// TIA Portal V16 export
// export: Created 2024-12-03T15:41:45.1410712Z, ExportSetting WithReadOnly, DisplayName Totally Integrated Automation Portal, DisplayVersion V16 Update 6, DisplayName TIA Portal Version Control Interface, DisplayVersion V16 Update 2, DisplayName TIA Portal Openness, DisplayVersion V16 Update 6, DisplayName TIA Portal Teamcenter Gateway, DisplayVersion V16, DisplayName SINAMICS Startdrive Advanced, DisplayVersion V16 Update 5, DisplayName SINAMICS Startdrive G130, G150, S120, S150, SINAMICS MV, S210, DisplayVersion V16 Update 5, DisplayName SINAMICS Startdrive G110M, G120, G120C, G120D, G120P, G115D, DisplayVersion V16 Update 5, DisplayName STEP 7 Professional, DisplayVersion V16 Update 6, DisplayName STEP 7 Safety, DisplayVersion V16, DisplayName WinCC Advanced / Unified PC, DisplayVersion V16 Update 6
TYPE "IT2000M_Scale_IN_UDT"
// stored: CreationDate 2021-07-13T07:41:36.2278727Z, InterfaceModifiedDate 2021-07-11T06:56:03.4750348Z, IsConsistent true, LibraryConformanceStatus The object is library-conformant., ModifiedDate 2021-07-11T06:56:03.4750348Z
   STRUCT
      Inputs : Struct
         spare : Byte;
         spare_0 : Bool;
         spare_1 : Bool;
         spare_2 : Bool;
         spare_3 : Bool;
         spare_4 : Bool;
         spare_5 : Bool;
         Input_E0 : Bool;
         Input_E1 : Bool;
      END_STRUCT;
      Outputs : Struct
         spare : Byte;
         spare_0 : Bool;
         spare_1 : Bool;
         spare_2 : Bool;
         spare_3 : Bool;
         spare_4 : Bool;
         spare_5 : Bool;
         Output_A0 : Bool;
         Output_A1 : Bool;
      END_STRUCT;
      NetWeight : Int;
      GrossWeight : Int;
      Status : Struct
         Handshake : Bool;
         Status : Bool;   // 1 = command carried out
         OutOfTolerance : Bool;
         FlowRateLow : Bool;
         spare_0 : Bool;
         spare_1 : Bool;
         spare_2 : Bool;
         ReadyForStart : Bool;
         GrossUnderZero : Bool;
         OverLoad : Bool;
         ScaleInMotion : Bool;
         Error : Bool;
         TrailingDecimals0 : Bool;
         TrailingDecimals1 : Bool;
         TrailingDecimals2 : Bool;
         WeightFactor10 : Bool;
      END_STRUCT;
      FillingStepCounter : Int;
      NetWeight_1 : Real;
      GrossWeight_1 : Real;
      StepperCounter : Int;
   END_STRUCT;
END_TYPE
